FUNCTION_BLOCK FB_ComponentT EXTENDS FB_Element
VAR_INPUT
END_VAR
VAR_OUTPUT
END_VAR
VAR
	bAbort: BOOL;
END_VAR

super^();

METHOD PROTECTED M_Execute : BOOL (* Return*)

IF bAbort THEN
	P_Event.M_Abort('msg', 0);
END_IF
END_METHOD

END_FUNCTION_BLOCK

(* stored: Version 1.1.0.1
   POU FB_ComponentT: Id {735f813a-3349-0a60-30db-82124ffd38eb}, SpecialFunc None
   Method M_Execute: Id {2088ebc2-7f48-06a1-0627-bd98553609ee} *)
